// TIA Portal V20 export
// export: Created 2026-08-13T15:37:27.6641289Z, ExportSetting WithDefaults, DisplayName Totally Integrated Automation Portal, DisplayVersion V20 Update 5, DisplayName TIA Portal Openness, DisplayVersion V20 Update 4, DisplayName TIA Portal Version Control Interface, DisplayVersion V20 Update 5, DisplayName SINAMICS Startdrive Advanced, DisplayVersion V20, DisplayName SINAMICS DCC, DisplayVersion V20, DisplayName SINAMICS Startdrive G130, G150, S120, S150, SINAMICS MV, G220, S200, S210, DisplayVersion V20, DisplayName SINAMICS Startdrive G110M, G120, G120C, G120D, G120P, G115D, DisplayVersion V20, DisplayName STEP 7 Professional, DisplayVersion V20 Update 5, DisplayName STEP 7 Safety, DisplayVersion V20 Update 2, DisplayName WinCC Basic/Comfort/Advanced, DisplayVersion V20 Update 5, DisplayName WinCC Unified, DisplayVersion V20 Update 5
DATA_BLOCK "iDB_HopperBlockageMonitor"   // DB51
VERSION : 0.1
// Single instance of FB_HopperBlockageMonitor (S6 request #1, hopper-blockage alarm). Members mirror the FB STATIC section; BlockedTimeThreshold (T#60S) and ClearDebounceTime (T#2S) carry the commissioning defaults (C-307/C-309). Hand-authored per the compile-error-playbook's synthesize-produced-FB path.
// stored: AutoNumber true, DBAccessibleFromOPCUA true, InstanceOfName FB_HopperBlockageMonitor, InstanceOfType FB
"FB_HopperBlockageMonitor"
   // VAR RETAIN
   //    IO { S7_SetPoint := 'True'} : "UDT_HopperBlockageIO";
   // END_VAR
   // VAR
   //    HighQualified : Bool;
   //    BlockActive : Bool;
   //    BlockActiveMem : Bool;
   //    PauseEdge : Bool;
   //    AccumulatedElapsed : Time;
   //    CumulativeElapsed : Time;
   //    ZeroTime : Time;
   //    ClearDebounceTimer { S7_SetPoint := 'True'} : TON_TIME;
   //    PersistenceTimer { S7_SetPoint := 'True'} : TON_TIME;
   // END_VAR
BEGIN
   IO.BlockedTimeThreshold := T#60S;
   IO.ClearDebounceTime := T#2S;
END_DATA_BLOCK
